// TIA Portal V16 export
// export: Created 2023-09-11T12:14:55.2039995Z, ExportSetting WithDefaults, DisplayName Totally Integrated Automation Portal, DisplayVersion V16 Update 6, DisplayName TIA Portal Version Control Interface, DisplayVersion V16 Update 2, DisplayName TIA Portal Openness, DisplayVersion V16 Update 6, DisplayName STEP 7 Professional, DisplayVersion V16 Update 6, DisplayName STEP 7 Safety, DisplayVersion V16, DisplayName WinCC Advanced, DisplayVersion V16 Update 6
FUNCTION "04_A_Convert_Scaling_analog" : Void   // FC14, LAD
TITLE = Funkcja konwertera analogów
{ S7_Optimized_Access := 'TRUE' }
AUTHOR : RTecmer
VERSION : 0.1
// Konwertowanie zmiennych procesowych
// stored: AutoNumber true, IsIECCheckEnabled false, SetENOAutomatically false, UDAEnableTagReadback false
BEGIN

REGION Network 1: Przepywomierz Q1 Pompownia
   // Pobrane z Modbus RTU
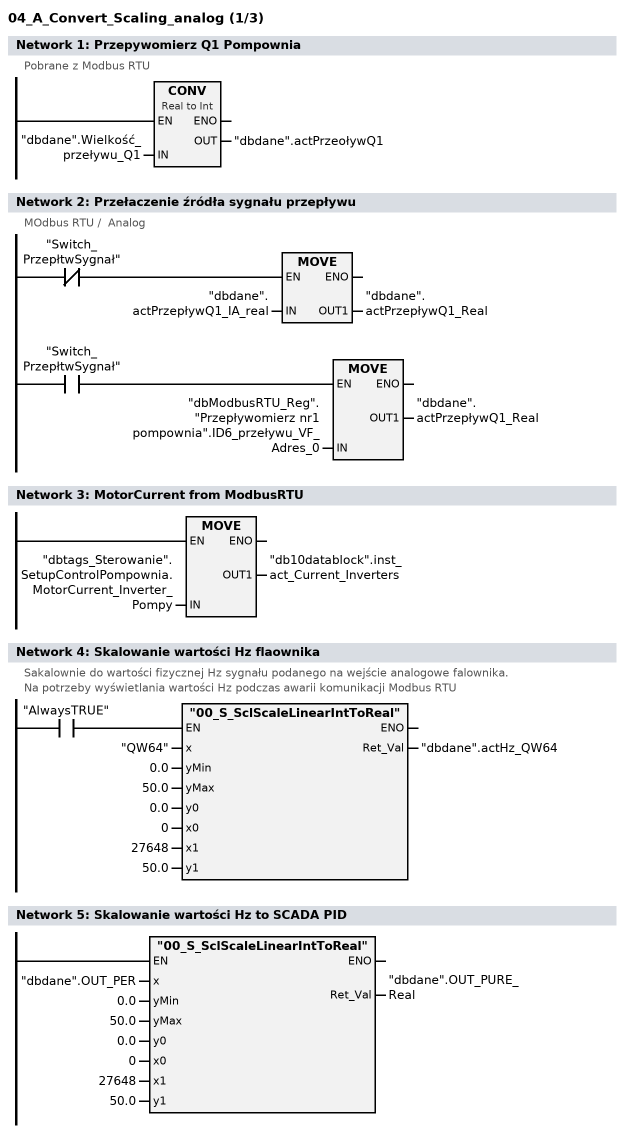
   RUNG wire#powerrail
      { S7_Templates := "[SrcType := Real, DestType := Int]" } Convert(in := "dbdane".Wielkość_przeływu_Q1, out => "dbdane".actPrzeoływQ1)
   END_RUNG
   // the same network as SCL:
   "dbdane".actPrzeoływQ1 := REAL_TO_INT("dbdane".Wielkość_przeływu_Q1);
END_REGION

REGION Network 2: Przełaczenie źródła sygnału przepływu
   // MOdbus RTU /  Analog
   RUNG wire#powerrail
      I_Contact( "Switch_PrzepłtwSygnał" )
      Move(in := "dbdane".actPrzepływQ1_IA_real, out1 => "dbdane".actPrzepływQ1_Real)
   END_RUNG
   RUNG wire#powerrail
      Contact( "Switch_PrzepłtwSygnał" )
      Move(in := "dbModbusRTU_Reg"."Przepływomierz nr1 pompownia".ID6_przeływu_VF_Adres_0, out1 => "dbdane".actPrzepływQ1_Real)
   END_RUNG
   // the same network as SCL:
   IF NOT "Switch_PrzepłtwSygnał" THEN "dbdane".actPrzepływQ1_Real := "dbdane".actPrzepływQ1_IA_real; END_IF;
   IF "Switch_PrzepłtwSygnał" THEN
       "dbdane".actPrzepływQ1_Real := "dbModbusRTU_Reg"."Przepływomierz nr1 pompownia".ID6_przeływu_VF_Adres_0;
   END_IF;
END_REGION

REGION Network 3: MotorCurrent from ModbusRTU
   RUNG wire#powerrail
      Move(in := "dbtags_Sterowanie".SetupControlPompownia.MotorCurrent_Inverter_Pompy, out1 => "db10datablock".inst_act_Current_Inverters)
   END_RUNG
   // the same network as SCL:
   "db10datablock".inst_act_Current_Inverters := "dbtags_Sterowanie".SetupControlPompownia.MotorCurrent_Inverter_Pompy;
END_REGION

REGION Network 4: Skalowanie wartości Hz flaownika
   // Sakalownie do wartości fizycznej Hz sygnału podanego na wejście analogowe falownika.
   // Na potrzeby wyświetlania wartości Hz podczas awarii komunikacji Modbus RTU
   RUNG wire#powerrail
      Contact( "AlwaysTRUE" )
      "00_S_SclScaleLinearIntToReal"(x := "QW64", yMin := 0.0, yMax := 50.0, y0 := 0.0, x0 := 0, x1 := 27648, y1 := 50.0, Ret_Val => "dbdane".actHz_QW64)
   END_RUNG
   // the same network as SCL:
   IF "AlwaysTRUE" THEN
       "dbdane".actHz_QW64 := "00_S_SclScaleLinearIntToReal"(x := "QW64",
                               yMin := 0.0,
                               yMax := 50.0,
                               y0 := 0.0,
                               x0 := 0,
                               x1 := 27648,
                               y1 := 50.0);
   END_IF;
END_REGION

REGION Network 5: Skalowanie wartości Hz to SCADA PID
   RUNG wire#powerrail
      "00_S_SclScaleLinearIntToReal"(x := "dbdane".OUT_PER, yMin := 0.0, yMax := 50.0, y0 := 0.0, x0 := 0, x1 := 27648, y1 := 50.0, Ret_Val => "dbdane".OUT_PURE_Real)
   END_RUNG
   // the same network as SCL:
   "dbdane".OUT_PURE_Real := "00_S_SclScaleLinearIntToReal"(x := "dbdane".OUT_PER,
                           yMin := 0.0,
                           yMax := 50.0,
                           y0 := 0.0,
                           x0 := 0,
                           x1 := 27648,
                           y1 := 50.0);
END_REGION

REGION Network 7: Ciśnienie kierunek miasto
   // Pomiar z czujnika B6 poziom "Przetłaczanie" - wylot za zasuwą
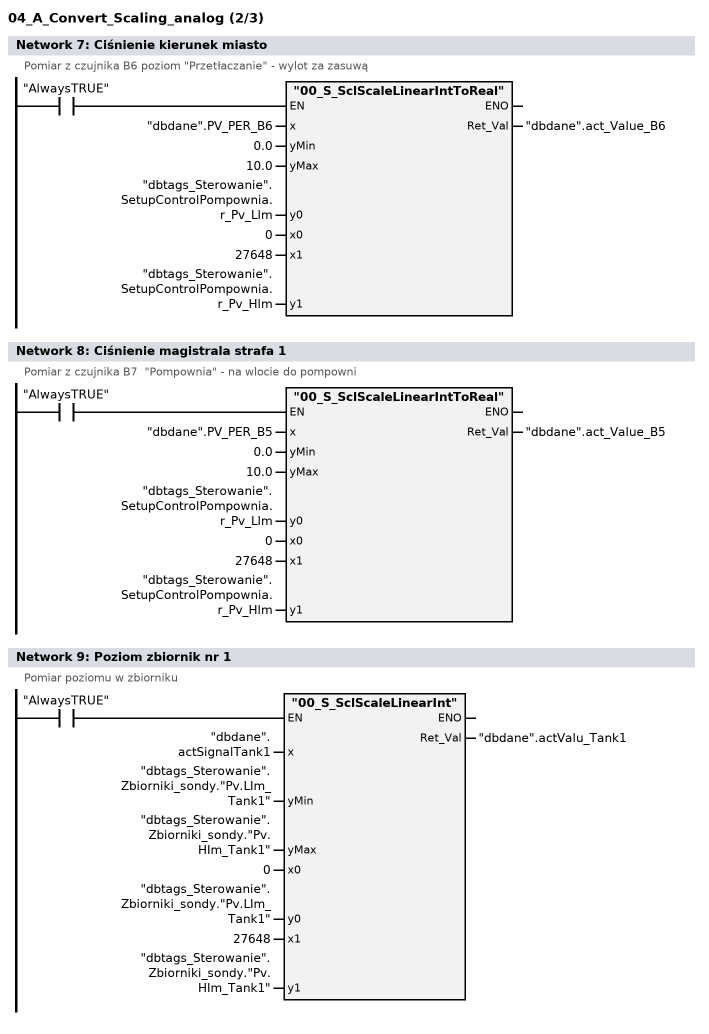
   RUNG wire#powerrail
      Contact( "AlwaysTRUE" )
      "00_S_SclScaleLinearIntToReal"(x := "dbdane".PV_PER_B6, yMin := 0.0, yMax := 10.0, y0 := "dbtags_Sterowanie".SetupControlPompownia.r_Pv_Llm, x0 := 0, x1 := 27648, y1 := "dbtags_Sterowanie".SetupControlPompownia.r_Pv_Hlm, Ret_Val => "dbdane".act_Value_B6)
   END_RUNG
   // the same network as SCL:
   IF "AlwaysTRUE" THEN
       "dbdane".act_Value_B6 := "00_S_SclScaleLinearIntToReal"(x := "dbdane".PV_PER_B6,
                               yMin := 0.0,
                               yMax := 10.0,
                               y0 := "dbtags_Sterowanie".SetupControlPompownia.r_Pv_Llm,
                               x0 := 0,
                               x1 := 27648,
                               y1 := "dbtags_Sterowanie".SetupControlPompownia.r_Pv_Hlm);
   END_IF;
END_REGION

REGION Network 8: Ciśnienie magistrala strafa 1
   // Pomiar z czujnika B7  "Pompownia" - na wlocie do pompowni
   RUNG wire#powerrail
      Contact( "AlwaysTRUE" )
      "00_S_SclScaleLinearIntToReal"(x := "dbdane".PV_PER_B5, yMin := 0.0, yMax := 10.0, y0 := "dbtags_Sterowanie".SetupControlPompownia.r_Pv_Llm, x0 := 0, x1 := 27648, y1 := "dbtags_Sterowanie".SetupControlPompownia.r_Pv_Hlm, Ret_Val => "dbdane".act_Value_B5)
   END_RUNG
   // the same network as SCL:
   IF "AlwaysTRUE" THEN
       "dbdane".act_Value_B5 := "00_S_SclScaleLinearIntToReal"(x := "dbdane".PV_PER_B5,
                               yMin := 0.0,
                               yMax := 10.0,
                               y0 := "dbtags_Sterowanie".SetupControlPompownia.r_Pv_Llm,
                               x0 := 0,
                               x1 := 27648,
                               y1 := "dbtags_Sterowanie".SetupControlPompownia.r_Pv_Hlm);
   END_IF;
END_REGION

REGION Network 9: Poziom zbiornik nr 1
   // Pomiar poziomu w zbiorniku
   RUNG wire#powerrail
      Contact( "AlwaysTRUE" )
      "00_S_SclScaleLinearInt"(x := "dbdane".actSignalTank1, yMin := "dbtags_Sterowanie".Zbiorniki_sondy."Pv.LIm_Tank1", yMax := "dbtags_Sterowanie".Zbiorniki_sondy."Pv.HIm_Tank1", x0 := 0, y0 := "dbtags_Sterowanie".Zbiorniki_sondy."Pv.LIm_Tank1", x1 := 27648, y1 := "dbtags_Sterowanie".Zbiorniki_sondy."Pv.HIm_Tank1", Ret_Val => "dbdane".actValu_Tank1)
   END_RUNG
   // the same network as SCL:
   IF "AlwaysTRUE" THEN
       "dbdane".actValu_Tank1 := "00_S_SclScaleLinearInt"(x := "dbdane".actSignalTank1,
                               yMin := "dbtags_Sterowanie".Zbiorniki_sondy."Pv.LIm_Tank1",
                               yMax := "dbtags_Sterowanie".Zbiorniki_sondy."Pv.HIm_Tank1",
                               x0 := 0,
                               y0 := "dbtags_Sterowanie".Zbiorniki_sondy."Pv.LIm_Tank1",
                               x1 := 27648,
                               y1 := "dbtags_Sterowanie".Zbiorniki_sondy."Pv.HIm_Tank1");
   END_IF;
END_REGION

REGION Network 10: Poziom zbiornik nr 2
   // Pomiar poziomu w zbiorniku
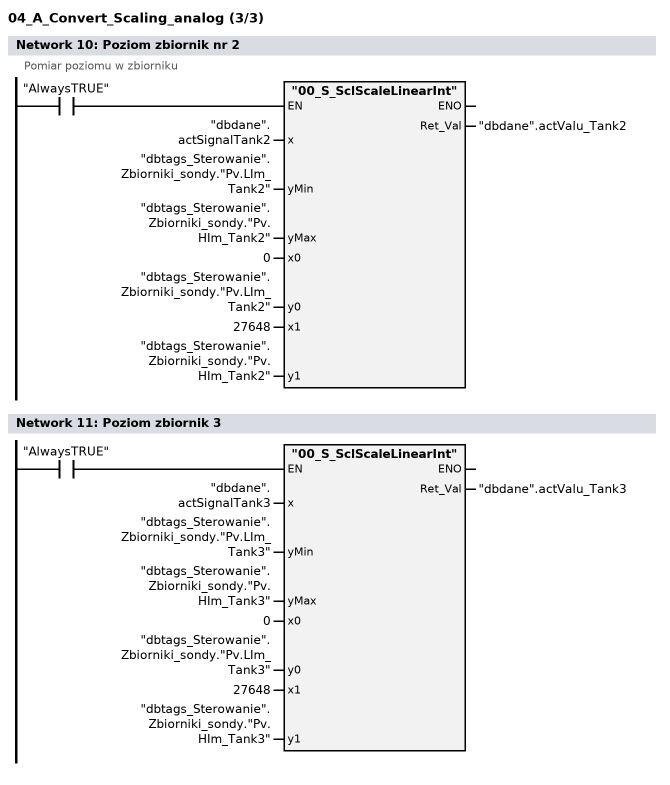
   RUNG wire#powerrail
      Contact( "AlwaysTRUE" )
      "00_S_SclScaleLinearInt"(x := "dbdane".actSignalTank2, yMin := "dbtags_Sterowanie".Zbiorniki_sondy."Pv.LIm_Tank2", yMax := "dbtags_Sterowanie".Zbiorniki_sondy."Pv.HIm_Tank2", x0 := 0, y0 := "dbtags_Sterowanie".Zbiorniki_sondy."Pv.LIm_Tank2", x1 := 27648, y1 := "dbtags_Sterowanie".Zbiorniki_sondy."Pv.HIm_Tank2", Ret_Val => "dbdane".actValu_Tank2)
   END_RUNG
   // the same network as SCL:
   IF "AlwaysTRUE" THEN
       "dbdane".actValu_Tank2 := "00_S_SclScaleLinearInt"(x := "dbdane".actSignalTank2,
                               yMin := "dbtags_Sterowanie".Zbiorniki_sondy."Pv.LIm_Tank2",
                               yMax := "dbtags_Sterowanie".Zbiorniki_sondy."Pv.HIm_Tank2",
                               x0 := 0,
                               y0 := "dbtags_Sterowanie".Zbiorniki_sondy."Pv.LIm_Tank2",
                               x1 := 27648,
                               y1 := "dbtags_Sterowanie".Zbiorniki_sondy."Pv.HIm_Tank2");
   END_IF;
END_REGION

REGION Network 11: Poziom zbiornik 3
   RUNG wire#powerrail
      Contact( "AlwaysTRUE" )
      "00_S_SclScaleLinearInt"(x := "dbdane".actSignalTank3, yMin := "dbtags_Sterowanie".Zbiorniki_sondy."Pv.LIm_Tank3", yMax := "dbtags_Sterowanie".Zbiorniki_sondy."Pv.HIm_Tank3", x0 := 0, y0 := "dbtags_Sterowanie".Zbiorniki_sondy."Pv.LIm_Tank3", x1 := 27648, y1 := "dbtags_Sterowanie".Zbiorniki_sondy."Pv.HIm_Tank3", Ret_Val => "dbdane".actValu_Tank3)
   END_RUNG
   // the same network as SCL:
   IF "AlwaysTRUE" THEN
       "dbdane".actValu_Tank3 := "00_S_SclScaleLinearInt"(x := "dbdane".actSignalTank3,
                               yMin := "dbtags_Sterowanie".Zbiorniki_sondy."Pv.LIm_Tank3",
                               yMax := "dbtags_Sterowanie".Zbiorniki_sondy."Pv.HIm_Tank3",
                               x0 := 0,
                               y0 := "dbtags_Sterowanie".Zbiorniki_sondy."Pv.LIm_Tank3",
                               x1 := 27648,
                               y1 := "dbtags_Sterowanie".Zbiorniki_sondy."Pv.HIm_Tank3");
   END_IF;
END_REGION
END_FUNCTION
